(* IEC 61131-3 sources: cc_kush_rewrite/Functions/Utilities, 5 files *)

(* ---- FC_MotorSyncronizedWork.st ---- *)
FUNCTION FC_MotorSyncronizedWork : BOOL
VAR_INPUT
	motor1 : ST_Motor;
	motor2 : ST_Motor;
END_VAR
VAR
END_VAR
FC_MotorSyncronizedWork := (
	// Контактор и ЧРП в работе у мотора 1
		motor1.fbStateKM.qxSignal
	AND	motor1.VFD.fbStateIsWorking.qxSignal
	// Контактор и ЧРП в работе у мотора 2
	AND	motor2.fbStateKM.qxSignal
	AND	motor2.VFD.fbStateIsWorking.qxSignal )
	// Частота мотора 1 и мотора 2 равны с учётом погрешности
	AND ( ABS(motor1.VFD.rActualFrequency - motor2.VFD.rActualFrequency) <= VFD_FREQUENCY_INACCURANCY );

END_FUNCTION

(* ---- FC_SwapBytesInWord.st ---- *)
FUNCTION FC_SwapBytesInWord : WORD
VAR_INPUT
    wInputValue : WORD;                         // Входное значение WORD
END_VAR
VAR
    uByteConverter : U_ByteToWord;              // Конвертер для работы с байтами
END_VAR

// Загружаем входное значение в конвертер
uByteConverter.wTag := wInputValue;

// Меняем местами байты: младший байт становится старшим, старший - младшим
FC_SwapBytesInWord := SHL(TO_WORD(uByteConverter.bTag[0]), 8) OR TO_WORD(uByteConverter.bTag[1]);

END_FUNCTION

(* ---- FC_SwapBytesInWordArray.st ---- *)
FUNCTION FC_SwapBytesInWordArray : ARRAY [0..1] OF WORD
VAR_INPUT
    awInputArray : ARRAY [0..1] OF WORD;        // Входной массив из двух WORD
END_VAR
VAR
    uByteConverter : U_ByteToWord;              // Конвертер для работы с байтами
    awOutputArray : ARRAY [0..1] OF WORD;       // Выходной массив
END_VAR

// Обработка первого WORD (индекс 0)
uByteConverter.wTag := awInputArray[0];
// Меняем местами байты и записываем в выходной массив
awOutputArray[0] := SHL(TO_WORD(uByteConverter.bTag[0]), 8) OR TO_WORD(uByteConverter.bTag[1]);

// Обработка второго WORD (индекс 1)
uByteConverter.wTag := awInputArray[1];
// Меняем местами байты и записываем в выходной массив
awOutputArray[1] := SHL(TO_WORD(uByteConverter.bTag[0]), 8) OR TO_WORD(uByteConverter.bTag[1]);

// Возвращаем преобразованный массив
FC_SwapBytesInWordArray := awOutputArray;

END_FUNCTION

(* ---- FC_SwapWordArrayElements.st ---- *)
FUNCTION FC_SwapWordArrayElements : ARRAY [0..1] OF WORD
VAR_INPUT
    awInputArray : ARRAY [0..1] OF WORD;        // Входной массив из двух WORD
END_VAR
VAR
    awOutputArray : ARRAY [0..1] OF WORD;       // Выходной массив
END_VAR
// Меняем местами элементы массива: [0] -> [1], [1] -> [0]
awOutputArray[0] := awInputArray[1];
awOutputArray[1] := awInputArray[0];

// Возвращаем массив с переставленными элементами
FC_SwapWordArrayElements := awOutputArray;

END_FUNCTION

(* ---- FC_VFD_ChangeReadMode.st ---- *)
FUNCTION FC_VFD_ChangeReadMode : BOOL
VAR_INPUT
	vfd : REFERENCE TO ST_VFD;
	mode : BOOL; // 0 - физический вход, 1 - Modbus
END_VAR
VAR
END_VAR
IF mode THEN
	vfd.rActualFrequency := vfd.uActualFrequency.rTag; // Чтение регистров ModbusRTU
ELSE
	vfd.rActualFrequency := vfd.fbActualFrequency.qrProcessedValue; // Чтение обработанного (масштабированного) аналогового сигнала с модуля
END_IF;

END_FUNCTION
